// TwinCAT 3 PLC project Tc3_Component
// Title: Tc3_Component
// Company: Zerlauth
// Author: Peter Zerlauth
// ProjectVersion: 0.0.0.0
// Description: ISA88 State Model with Observer and Events
// ProgramVersion: 3.1.4024.0
// libraries:
//   Tc2_Standard, * (Beckhoff Automation GmbH)
//   Tc2_System, * (Beckhoff Automation GmbH)
//   Tc2_Utilities, * (Beckhoff Automation GmbH)
// project tree:
//   Component/Event/ E_Event.TcDUT (not stored), E_Behaviour.TcDUT (not stored), FB_Event.TcPOU, I_Event.TcIO (not stored), ST_Event.TcDUT
//   Component/ E_Request.TcDUT, E_State.TcDUT (not stored), FB_Component.TcPOU (not stored), I_Component.TcIO
//   Component/Info/ FB_Info.TcPOU (not stored), I_Info.TcIO (not stored)
//   Component/Observer/ FB_Observer.TcPOU, I_Observer.TcIO
//   CyclicCall/ FB_Cycle.TcPOU (not stored), I_Cycle.TcIO (not stored)
//   IO/ DigitalInput.TcPOU (not stored), AnalogInput.TcPOU (not stored), DigitalOutput.TcPOU (not stored), AnalogOutput.TcPOU (not stored), I_Channel.TcIO, I_DigitalInput.TcIO, I_AnalogInput.TcIO, I_DigitalOutput.TcIO (not stored), I_AnalogOutput.TcIO
//   List/ FB_ListComponent.TcPOU, FB_ListObject.TcPOU (not stored), FB_ListString.TcPOU (not stored), I_ListComponent.TcIO, I_ListObject.TcIO (not stored), I_ListString.TcIO (not stored)
//   Logger/ FB_LoggerFactory.TcPOU, I_Logger.TcIO (not stored)
//   Object/ I_Object.TcIO (not stored)
//   Sequence/ FB_Sequence.TcPOU (not stored), I_Sequence.TcIO
// (motion and I/O tree: see PLC project example)
// real-time tasks:
//   TASK plcTask1: cycle T#25000us, priority 20, ADS port 350

// ---- Component/Event/ST_Event.TcDUT
TYPE ST_Event :
STRUCT
	Source:			I_Component;
	Instance:		STRING(255);
	Class:			STRING(255);
	EventType:		E_Event;
	Timestamp:   	ULINT;
	ID:				UDINT;
	Message:		STRING(255);
	Arguments:		STRING(255);
	Active:			BOOL;
	New:			BOOL;
END_STRUCT
END_TYPE

// ---- Component/E_Request.TcDUT
{attribute 'qualified_only'}
{attribute 'strict'}
{attribute 'to_string'}
TYPE E_Request :
(
	{attribute 'hide'}
    Undefined   := 0,
	Reset       := 1,
    Start       := 2,
    Pause       := 4,	
    Hold      	:= 8,
	Complete	:= 16,	
    Stop        := 32,
	Abort       := 64
);
END_TYPE

// ---- Component/I_Component.TcIO
INTERFACE I_Component EXTENDS I_Cycle

METHOD PUBLIC M_OnNotify
VAR_INPUT
	eState:				E_State;
END_VAR
END_METHOD

METHOD PUBLIC M_Request : BOOL
VAR_INPUT
	eRequest:	E_Request;
END_VAR
END_METHOD

PROPERTY PUBLIC P_Event : I_Event
GET
END_GET
END_PROPERTY

PROPERTY PUBLIC P_Info : I_Info
GET
END_GET
END_PROPERTY

PROPERTY PUBLIC P_Observer : I_Observer
GET
END_GET
END_PROPERTY

PROPERTY PUBLIC P_State : E_State
GET
END_GET
END_PROPERTY

END_INTERFACE

// ---- Component/Observer/I_Observer.TcIO
INTERFACE I_Observer

METHOD M_Attach : BOOL
VAR_INPUT
	Object: 	I_Component;
END_VAR
END_METHOD

METHOD M_Detach : BOOL
VAR_INPUT
	Object: 	I_Component;
END_VAR
END_METHOD

METHOD M_Notify : BOOL
VAR_INPUT
	eState:				E_State;
END_VAR
END_METHOD

END_INTERFACE

// ---- IO/I_Channel.TcIO
INTERFACE I_Channel EXTENDS I_Object

PROPERTY PUBLIC P_ID : String(25)
GET
END_GET
END_PROPERTY

END_INTERFACE

// ---- IO/I_DigitalInput.TcIO
INTERFACE I_DigitalInput EXTENDS I_Channel

PROPERTY P_Value : bool
GET
END_GET
END_PROPERTY

END_INTERFACE

// ---- IO/I_AnalogInput.TcIO
INTERFACE I_AnalogInput EXTENDS I_Channel

PROPERTY P_Value : LREAL
GET
END_GET
END_PROPERTY

END_INTERFACE

// ---- IO/I_AnalogOutput.TcIO
INTERFACE I_AnalogOutput EXTENDS I_Channel

PROPERTY P_Value : LREAL
SET
END_SET
END_PROPERTY

END_INTERFACE

// ---- List/I_ListComponent.TcIO
INTERFACE I_ListComponent

METHOD PUBLIC M_Add : BOOL
VAR_INPUT
	Object: 	I_Component;
END_VAR
END_METHOD

METHOD PUBLIC M_Clear : BOOL
END_METHOD

METHOD PUBLIC M_Find : DINT
VAR_INPUT
	Object: 	I_Component;
END_VAR
END_METHOD

METHOD PUBLIC M_Index : I_Component
VAR_INPUT
	Index: 	DINT;
END_VAR
END_METHOD

METHOD PUBLIC M_Remove : BOOL
VAR_INPUT
	Object: 	I_Component;
END_VAR
END_METHOD

METHOD PUBLIC M_Request : BOOL
VAR_INPUT
	eRequest:		E_Request;
END_VAR
END_METHOD

PROPERTY P_Length : DINT
GET
END_GET
END_PROPERTY

END_INTERFACE

// ---- Sequence/I_Sequence.TcIO
INTERFACE I_Sequence EXTENDS I_Object

METHOD PUBLIC M_Await 
VAR_INPUT
	Message:				STRING(255);
	tTimeout:				TIME;
	bCondition:				BOOL;
	nNumber:				INT;	
END_VAR
END_METHOD

END_INTERFACE

// ---- Component/Event/FB_Event.TcPOU
FUNCTION_BLOCK FB_Event EXTENDS FB_ListString IMPLEMENTS I_Event
VAR_INPUT
	bIngoreHold:			BOOL:= TRUE;
	bIngorePause:			BOOL:= TRUE;
END_VAR
VAR_OUTPUT
END_VAR
VAR
	iParent:			I_Component;
	iLogger:			I_Logger;
	stError:			ST_Event;
	stWarning:			ST_Event;
	stInformation:		ST_Event;
	stDebug:			ST_Event;
END_VAR

SUPER^();

METHOD FB_init : BOOL
VAR_INPUT
	bInitRetains : BOOL; // if TRUE, the retain variables are initialized (warm start / cold start)
	bInCopyCode : BOOL;  // if TRUE, the instance afterwards gets moved into the copy code (online change)
	iParent:			I_Component;
END_VAR
THIS^.iParent:= iParent;
END_METHOD

METHOD INTERNAL M_Arguments : STRING(255)
VAR_INPUT
END_VAR
VAR
	nIndex:			INT;
END_VAR
WHILE nIndex < nLength DO
	M_Arguments:= Concat(Concat(M_Arguments, pList[nIndex]), '$N');
	nIndex:= nIndex + 1;
END_WHILE
END_METHOD

METHOD PUBLIC M_Debug : BOOL
VAR_INPUT
	Message:				STRING(255);
END_VAR
IF stDebug.Message <> Message THEN
	stDebug.New:= TRUE;
ELSE
	stDebug.New:= FALSE;
END_IF

stDebug.Source:= iParent;
stDebug.Instance:= iParent.P_Info.P_Instance;
stDebug.Class:= iParent.P_Info.P_Class;
stDebug.EventType:= E_Event.Debug;
stDebug.Timestamp:= F_GetSystemTime();
stDebug.ID:= 0;
stDebug.Message:= Message;
stDebug.Arguments:= M_Arguments();
stDebug.Active:= TRUE;

IF iLogger <> 0 THEN
	iLogger.M_Log(stDebug);
END_IF

M_Clear();
END_METHOD

METHOD PUBLIC M_Error : BOOL
VAR_INPUT
	Message:				STRING(255);
	ID:						UDINT;
	Behaviour:				E_Behaviour;
END_VAR
IF stError.Message <> Message THEN
	stError.Source:= iParent;
	stError.Instance:= iParent.P_Info.P_Instance;
	stError.Class:= iParent.P_Info.P_Class;
	stError.EventType:= E_Event.Error;
	stError.Timestamp:= F_GetSystemTime();
	stError.ID:= ID;
	stError.Message:= Message;
	stError.Arguments:= M_Arguments();
	stError.New:= TRUE;
	stError.Active:= TRUE;


	IF Behaviour >= E_Behaviour.Abort THEN
		iParent.M_Request(E_Request.Abort);
	ELSIF Behaviour >= E_Behaviour.Stop THEN
		iParent.M_Request(E_Request.Stop);
	ELSIF Behaviour >= E_Behaviour.Complete THEN	
		iParent.M_Request(E_Request.Complete);
	ELSIF Behaviour >= E_Behaviour.Hold THEN
		iParent.M_Request(E_Request.Hold);
	ELSIF Behaviour >= E_Behaviour.Pause THEN
		iParent.M_Request(E_Request.Pause);
	END_IF
	
	IF iLogger <> 0 THEN
		iLogger.M_Log(stError);
	END_IF
END_IF

M_Clear();
END_METHOD

METHOD PUBLIC M_Information : BOOL
VAR_INPUT
	Message:				STRING(255);
	ID:						UDINT;
END_VAR
IF stInformation.Message <> Message THEN
	stInformation.New:= TRUE;
ELSE
	stInformation.New:= FALSE;
END_IF

stInformation.Source:= iParent;
stInformation.Instance:= iParent.P_Info.P_Instance;
stInformation.Class:= iParent.P_Info.P_Class;
stInformation.EventType:= E_Event.Information;
stInformation.Timestamp:= F_GetSystemTime();
stInformation.ID:= ID;
stInformation.Message:= Message;
stInformation.Arguments:= M_Arguments();
stInformation.Active:= TRUE;

IF iLogger <> 0 THEN
	iLogger.M_Log(stInformation);
END_IF

M_Clear();
END_METHOD

METHOD PUBLIC M_Reset
VAR_INPUT
END_VAR
Memset(ADR(stError), 0, SIZEOF(stError));
Memset(ADR(stWarning), 0, SIZEOF(stWarning));
Memset(ADR(stInformation), 0, SIZEOF(stInformation));
Memset(ADR(stDebug), 0, SIZEOF(stDebug));
END_METHOD

METHOD PUBLIC M_Warning : BOOL
VAR_INPUT
	Message:				STRING(255);
	ID:						UDINT;
END_VAR
IF stWarning.Message <> Message THEN
	stWarning.New:= TRUE;
ELSE
	stWarning.New:= FALSE;
END_IF

stWarning.Source:= iParent;
stWarning.Instance:= iParent.P_Info.P_Instance;
stWarning.Class:= iParent.P_Info.P_Class;
stWarning.EventType:= E_Event.Warning;
stWarning.Timestamp:= F_GetSystemTime();
stWarning.ID:= ID;
stWarning.Message:= Message;
stWarning.Arguments:= M_Arguments();
stWarning.Active:= TRUE;

IF iLogger <> 0 THEN
	iLogger.M_Log(stWarning);
END_IF

M_Clear();
END_METHOD

PROPERTY PUBLIC P_Logger : I_Logger
GET
P_Logger:= iLogger;
END_GET
SET
iLogger:= P_Logger;
END_SET
END_PROPERTY

END_FUNCTION_BLOCK

// ---- Component/Observer/FB_Observer.TcPOU
{attribute 'no_explicit_call'} 
FUNCTION_BLOCK PUBLIC FB_Observer IMPLEMENTS I_Observer
VAR
	pList: 			POINTER TO I_Component;
	nLength:		DINT;
	{attribute 'conditionalshow'}
	aList:			POINTER TO POINTER TO ARRAY [0..100] OF I_Component:=ADR(pList);
END_VAR

METHOD FB_exit : BOOL
VAR_INPUT
	bInCopyCode : BOOL; // if TRUE, the exit method is called for exiting an instance that is copied afterwards (online change).
END_VAR
M_Clear();
END_METHOD

METHOD M_Attach : BOOL
VAR_INPUT
	Object: 	I_Component;
END_VAR
VAR
	pOldList: 	POINTER TO I_Component;
END_VAR
IF Object <> 0 THEN
	// First Item
	IF pList = 0 THEN
		nLength:= nLength + 1;
		pList:= __NEW(POINTER TO I_Component,DINT_TO_UDINT(nLength));
	ELSE
		// Item already in List
		IF M_Find(Object) = -1 THEN
			// backup 
			pOldList:= pList;
			// new Length
			nLength:= nLength + 1;
			// new pointer
			pList:= __NEW(POINTER TO I_Component,DINT_TO_UDINT(nLength));
			// restore
			Memcpy(pList,pOldList, SIZEOF(POINTER TO I_Component)*DINT_TO_UDINT(nLength -1));
			// delete old
			__DELETE(pOldList);
		ELSE
			M_Attach:= FALSE;	
			RETURN;
		END_IF
	END_IF
	IF pList = 0 THEN
		RETURN;
	END_IF
	// add new Object
	pList[nLength-1]:= Object;
	M_Attach:= TRUE;
ELSE
	M_Attach:= FALSE;	
END_IF
END_METHOD

METHOD M_Clear
IF pList <> 0 THEN
	nLength:= 0;
	__DELETE(pList);
END_IF
END_METHOD

METHOD M_Detach : BOOL
VAR_INPUT
	Object: 	I_Component;
END_VAR
VAR
	pOldList:			POINTER TO I_Component;
	nPosition: 			DINT;
END_VAR
IF Object <> 0 THEN
	// First Item
	IF nLength >= 0 THEN
		// Item already in List
		nPosition:= M_Find(Object);
		IF nPosition <> -1 THEN
			// backup 
			pOldList:= pList;
			// new Length
			nLength:= nLength -1;
			// new pointer
			pList:= __NEW(POINTER TO I_Component,DINT_TO_UDINT(nLength));
			// restore lower part
			Memcpy(pList,pOldList, SIZEOF(POINTER TO I_Component) * DINT_TO_UDINT(nPosition));
			//pList[nPosition]:= iObject;
			Memcpy(pList + (SIZEOF(POINTER TO I_Component)*nPosition),pOldList + (SIZEOF(POINTER TO I_Component)*(nPosition + 1)), SIZEOF(POINTER TO I_Component) * DINT_TO_UDINT(nLength - nPosition));
			// delete old
			__DELETE(pOldList);
		ELSE
			M_Detach:= FALSE;	
			RETURN;
		END_IF
	ELSE
		M_Detach:= FALSE;	
		RETURN;
	END_IF
	M_Detach:= TRUE;
ELSE
	M_Detach:= FALSE;	
END_IF
END_METHOD

METHOD M_Find : DINT
VAR_INPUT
	Object: 	I_Component;
END_VAR
VAR
	nIndex: 	UINT;
END_VAR
// Object already in List
M_Find := -1;
WHILE nIndex < nLength DO
    IF (pList[nIndex] = Object) THEN
        M_Find := nIndex;
        RETURN;
    END_IF
	nIndex := nIndex + 1;
END_WHILE
END_METHOD

METHOD M_Index : I_Component
VAR_INPUT
	Index: 	DINT;
END_VAR
IF Index <= nLength THEN
	M_Index:= pList[Index];
END_IF
END_METHOD

METHOD M_Notify : BOOL
VAR_INPUT
	eState:				E_State;
END_VAR

VAR
	nIndex: 	INT;
END_VAR
WHILE nIndex < nLength DO
	pList[nIndex].M_OnNotify(eState);
	nIndex:= nIndex + 1; 
END_WHILE
END_METHOD

PROPERTY P_Length : DINT
GET
P_Length:= nLength;
END_GET
END_PROPERTY

END_FUNCTION_BLOCK

// ---- List/FB_ListComponent.TcPOU
{attribute 'no_explicit_call'} 
FUNCTION_BLOCK FB_ListComponent IMPLEMENTS I_ListComponent
VAR
	nLength:		DINT;
	pList: 			POINTER TO I_Component;
	{attribute 'conditionalshow'}
	aList:			POINTER TO POINTER TO ARRAY [0..100] OF I_Component:=ADR(pList);
END_VAR

METHOD FB_exit : BOOL
VAR_INPUT
	bInCopyCode : BOOL; // if TRUE, the exit method is called for exiting an instance that is copied afterwards (online change).
END_VAR
M_Clear();
END_METHOD

METHOD PUBLIC M_Add : BOOL
VAR_INPUT
	Object: 	I_Component;
END_VAR
VAR
	pOldList: 	POINTER TO I_Component;
END_VAR
IF Object <> 0 THEN
	// First Item
	IF pList = 0 THEN
		nLength:= nLength + 1;
		pList:= __NEW(POINTER TO I_Component,DINT_TO_UDINT(nLength));
	ELSE
		// Item already in List
		IF M_Find(Object) = -1 THEN
			// backup 
			pOldList:= pList;
			// new Length
			nLength:= nLength + 1;
			// new pointer
			pList:= __NEW(POINTER TO I_Component,DINT_TO_UDINT(nLength));
			// restore
			Memcpy(pList,pOldList, SIZEOF(POINTER TO I_Component)*DINT_TO_UDINT(nLength -1));
			// delete old
			__DELETE(pOldList);
		ELSE
			M_Add:= FALSE;	
			RETURN;
		END_IF
	END_IF
	IF pList = 0 THEN
		RETURN;
	END_IF
	// add new Object
	pList[nLength-1]:= Object;
	M_Add:= TRUE;
ELSE
	M_Add:= FALSE;	
END_IF
END_METHOD

METHOD PUBLIC M_Clear : BOOL
// Clear
IF pList <> 0 THEN
	nLength:= 0;
	__DELETE(pList);
END_IF
M_Clear:= TRUE;
END_METHOD

METHOD PUBLIC M_Find : DINT
VAR_INPUT
	Object: 	I_Component;
END_VAR
VAR
	nIndex: 	UINT;
END_VAR
// Find
M_Find := -1;
WHILE nIndex < nLength DO
    IF (pList[nIndex] = Object) THEN
        M_Find := nIndex;
        RETURN;
    END_IF
	nIndex := nIndex + 1;
END_WHILE
END_METHOD

METHOD PUBLIC M_Index : I_Component
VAR_INPUT
	Index: 	DINT;
END_VAR
// Index
IF Index <= nLength THEN
	M_Index:= pList[Index];
END_IF
END_METHOD

METHOD PUBLIC M_Remove : BOOL
VAR_INPUT
	Object: 	I_Component;
END_VAR
VAR
	pOldList:			POINTER TO I_Component;
	nPosition: 			DINT;
END_VAR
// Remove
IF Object <> 0 THEN
	// First Item
	IF nLength >= 0 THEN
		// Item already in List
		nPosition:= M_Find(Object);
		IF nPosition <> -1 THEN
			// backup 
			pOldList:= pList;
			// new Length
			nLength:= nLength -1;
			// new pointer
			pList:= __NEW(POINTER TO I_Component,DINT_TO_UDINT(nLength));
			// restore lower part
			Memcpy(pList,pOldList, SIZEOF(POINTER TO I_Object) * DINT_TO_UDINT(nPosition));
			//pList[nPosition]:= iObject;
			Memcpy(pList + (SIZEOF(POINTER TO I_Component)*nPosition),pOldList + (SIZEOF(POINTER TO I_Component)*(nPosition + 1)), SIZEOF(POINTER TO I_Component) * DINT_TO_UDINT(nLength - nPosition));
			// delete old
			__DELETE(pOldList);
		ELSE
			M_Remove:= FALSE;	
			RETURN;
		END_IF
	ELSE
		M_Remove:= FALSE;	
		RETURN;
	END_IF
	M_Remove:= TRUE;
ELSE
	M_Remove:= FALSE;	
END_IF
END_METHOD

METHOD PUBLIC M_Request : BOOL
VAR_INPUT
	eRequest:		E_Request;
END_VAR
VAR
	nIndex:			INT:= 0;
END_VAR
// Request
M_Request:= TRUE;
WHILE nIndex < P_Length DO
	M_Request:= M_Request AND M_Index(nIndex).M_Request(eRequest);
	nIndex:= nIndex + 1;
END_WHILE
END_METHOD

PROPERTY PUBLIC P_Length : DINT
GET
P_Length:= nLength;
END_GET
END_PROPERTY

END_FUNCTION_BLOCK

// ---- Logger/FB_LoggerFactory.TcPOU
{attribute 'no_explicit_call'} 
FUNCTION_BLOCK FB_LoggerFactory IMPLEMENTS I_Logger
VAR
	pList: 			POINTER TO I_Logger;
	nLength:		DINT;
	{attribute 'conditionalshow'}
	aList:			POINTER TO POINTER TO ARRAY [0..100] OF I_Logger:=ADR(pList);
END_VAR

METHOD FB_exit : BOOL
VAR_INPUT
	bInCopyCode : BOOL; // if TRUE, the exit method is called for exiting an instance that is copied afterwards (online change).
END_VAR
M_Clear();
END_METHOD

METHOD M_Add : BOOL
VAR_INPUT
	Object: 	I_Logger;
END_VAR
VAR
	pOldList: 	POINTER TO I_Logger;
END_VAR
IF Object <> 0 THEN
	// First Item
	IF pList = 0 THEN
		nLength:= nLength + 1;
		pList:= __NEW(POINTER TO I_Logger,DINT_TO_UDINT(nLength));
	ELSE
		// Item already in List
		IF M_Find(Object) = -1 THEN
			// backup 
			pOldList:= pList;
			// new Length
			nLength:= nLength + 1;
			// new pointer
			pList:= __NEW(POINTER TO I_Object,DINT_TO_UDINT(nLength));
			// restore
			Memcpy(pList,pOldList, SIZEOF(POINTER TO I_Logger)*DINT_TO_UDINT(nLength -1));
			// delete old
			__DELETE(pOldList);
		ELSE
			M_Add:= FALSE;	
			RETURN;
		END_IF
	END_IF
	IF pList = 0 THEN
		RETURN;
	END_IF
	// add new Object
	pList[nLength-1]:= Object;
	M_Add:= TRUE;
ELSE
	M_Add:= FALSE;	
END_IF
END_METHOD

METHOD M_Clear : bool
IF pList <> 0 THEN
	nLength:= 0;
	__DELETE(pList);
END_IF
M_Clear:= True;
END_METHOD

METHOD M_Find : DINT
VAR_INPUT
	Object: 	I_Logger;
END_VAR
VAR
	nIndex: 	UINT;
END_VAR
// Object already in List
M_Find := -1;
WHILE nIndex < nLength DO
    IF (pList[nIndex] = Object) THEN
        M_Find := nIndex;
        RETURN;
    END_IF
	nIndex := nIndex + 1;
END_WHILE
END_METHOD

METHOD M_Index : I_Logger
VAR_INPUT
	Index: 	DINT;
END_VAR
IF Index <= nLength THEN
	M_Index:= pList[Index];
END_IF
END_METHOD

METHOD PUBLIC M_Log
VAR_INPUT
	stEvent:		ST_Event;
END_VAR
VAR
	nIndex: INT;
END_VAR
WHILE nIndex < nLength DO
	M_Index(nIndex).M_Log(stEvent);
	nIndex:= nIndex +1;
END_WHILE
END_METHOD

METHOD M_Remove : BOOL
VAR_INPUT
	Object: 	I_Logger;
END_VAR
VAR
	pOldList:			POINTER TO I_Logger;
	nPosition: 			DINT;
END_VAR
IF Object <> 0 THEN
	// First Item
	IF nLength >= 0 THEN
		// Item already in List
		nPosition:= M_Find(Object);
		IF nPosition <> -1 THEN
			// backup 
			pOldList:= pList;
			// new Length
			nLength:= nLength -1;
			// new pointer
			pList:= __NEW(POINTER TO I_Logger,DINT_TO_UDINT(nLength));
			// restore lower part
			Memcpy(pList,pOldList, SIZEOF(POINTER TO I_Logger) * DINT_TO_UDINT(nPosition));
			//pList[nPosition]:= iObject;
			Memcpy(pList + (SIZEOF(POINTER TO I_Logger)*nPosition),pOldList + (SIZEOF(POINTER TO I_Logger)*(nPosition + 1)), SIZEOF(POINTER TO I_Logger) * DINT_TO_UDINT(nLength - nPosition));
			// delete old
			__DELETE(pOldList);
		ELSE
			M_Remove:= FALSE;	
			RETURN;
		END_IF
	ELSE
		M_Remove:= FALSE;	
		RETURN;
	END_IF
	M_Remove:= TRUE;
ELSE
	M_Remove:= FALSE;	
END_IF
END_METHOD

PROPERTY P_Length : DINT
GET
P_Length:= nLength;
END_GET
END_PROPERTY

END_FUNCTION_BLOCK
